TYPE ST_XTS_TRANSPORT_CTRL :
STRUCT
  Cmd       : E_XTS_TRANSPORT_CTRL;
END_STRUCT
END_TYPE

(* stored: Version 1.1.0.1, ProductVersion 3.1.4024.12
   DUT ST_XTS_TRANSPORT_CTRL: Id {6f7582bd-8409-47a5-a9e3-2a3e50c13607} *)
